INTERFACE I_WORD EXTENDS I_Datatype

PROPERTY PUBLIC Value : REFERENCE TO WORD
GET
END_GET
END_PROPERTY

END_INTERFACE

(* stored: Version 1.1.0.1, ProductVersion 3.1.4024.15
   Itf I_WORD: Id {12953f6f-c677-0171-01cf-a725151d12a2}
   Property Value: Id {0faffda8-b0fa-03f8-2aa2-dee502b4be97}
   Get Get: Id {cd541c80-35cf-0ed9-3017-d228baba1d1b} *)
